(* PLC project AHU-Project.project, CODESYS CODESYS V3.5 SP21 Patch 5 *)
(* stored: creationDateTime 2026-06-15T00:53:37.6584983, modificationDateTime 2026-06-15T00:41:05.8983208 *)

PROGRAM PLC_PRG_LD
  VAR
    temp_LowerLimit : REAL;
    temp_UpperLimit : REAL;
    temp_SetCond : BOOL;
    temp_ResetCond : BOOL;
    RS_HeatControl : RS;
  END_VAR
  VAR  (* added by the conversion: wires and edge detectors of the diagram *)
    _SUB53_EN : BOOL;
  END_VAR

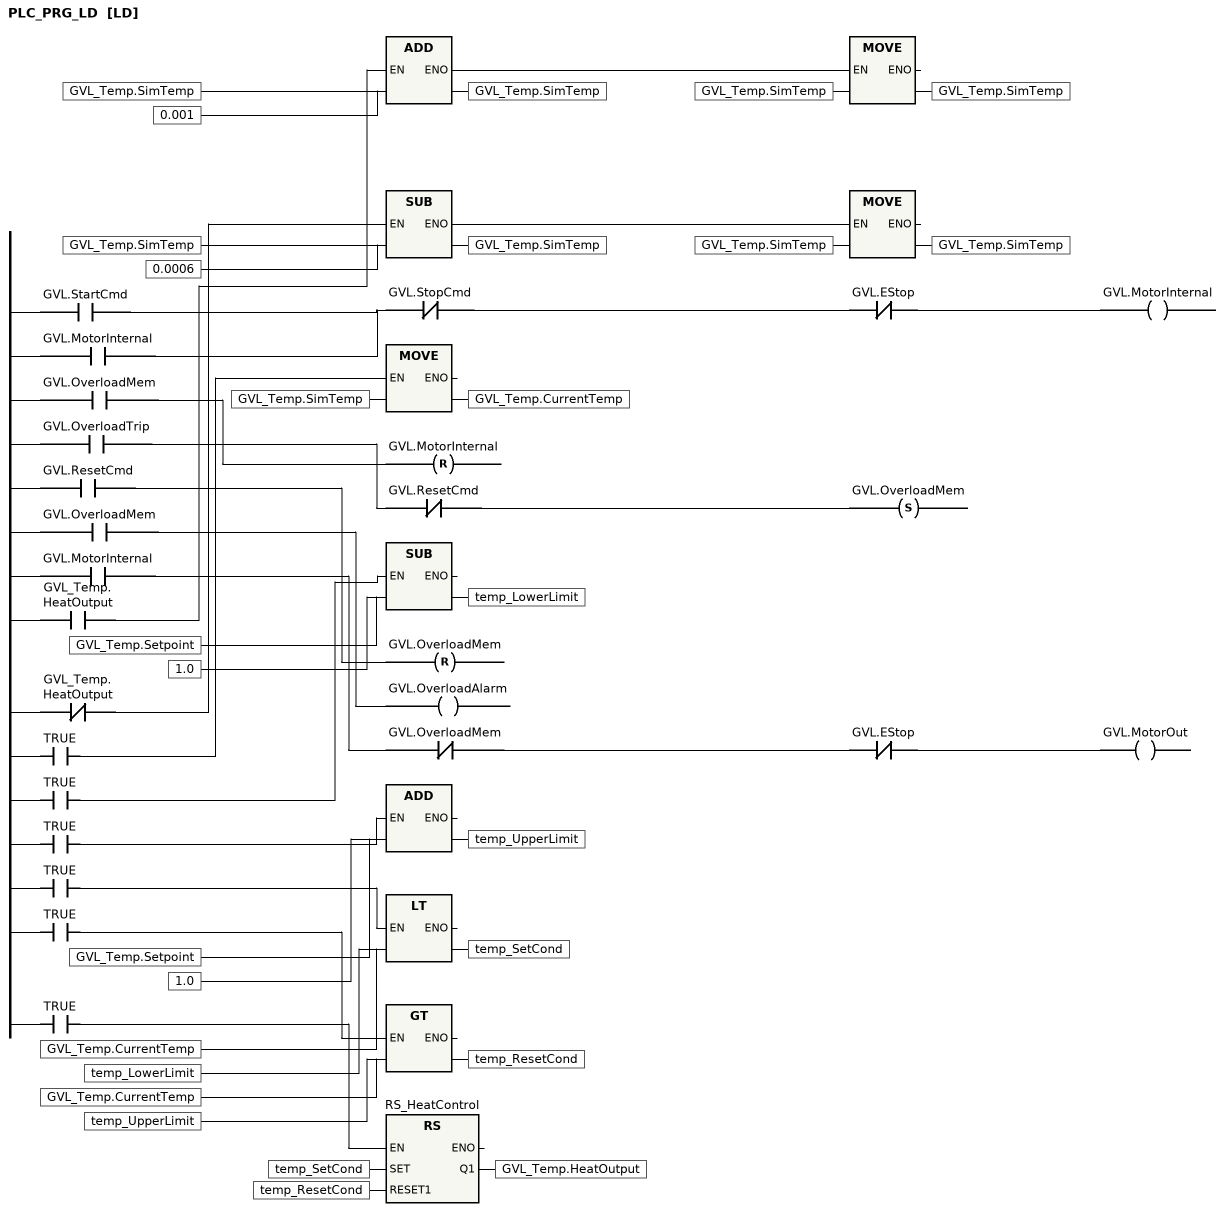
(* LD diagram, written out as Structured Text *)

GVL.MotorInternal := (GVL.StartCmd OR GVL.MotorInternal) AND NOT GVL.StopCmd AND NOT GVL.EStop;

IF GVL.OverloadMem THEN GVL.MotorInternal := FALSE; END_IF;

IF GVL.OverloadTrip AND NOT GVL.ResetCmd THEN GVL.OverloadMem := TRUE; END_IF;

IF GVL.ResetCmd THEN GVL.OverloadMem := FALSE; END_IF;

GVL.OverloadAlarm := GVL.OverloadMem;

GVL.MotorOut := GVL.MotorInternal AND NOT GVL.OverloadMem AND NOT GVL.EStop;

IF GVL_Temp.HeatOutput THEN GVL_Temp.SimTemp := GVL_Temp.SimTemp + 0.001; END_IF;
IF GVL_Temp.HeatOutput THEN GVL_Temp.SimTemp := GVL_Temp.SimTemp; END_IF;

_SUB53_EN := NOT GVL_Temp.HeatOutput;
IF _SUB53_EN THEN GVL_Temp.SimTemp := GVL_Temp.SimTemp - 0.0006; END_IF;
IF _SUB53_EN THEN GVL_Temp.SimTemp := GVL_Temp.SimTemp; END_IF;

IF TRUE THEN GVL_Temp.CurrentTemp := GVL_Temp.SimTemp; END_IF;

IF TRUE THEN temp_LowerLimit := GVL_Temp.Setpoint - 1.0; END_IF;

IF TRUE THEN temp_UpperLimit := GVL_Temp.Setpoint + 1.0; END_IF;

IF TRUE THEN temp_SetCond := GVL_Temp.CurrentTemp < temp_LowerLimit; END_IF;

IF TRUE THEN temp_ResetCond := GVL_Temp.CurrentTemp > temp_UpperLimit; END_IF;

RS_HeatControl(EN := TRUE, SET := temp_SetCond, RESET1 := temp_ResetCond, Q1 => GVL_Temp.HeatOutput);
END_PROGRAM
